Fanuc KAREL source: KT00074.KL

PROGRAM KT00074
%NOLOCKGROUP
VAR
  R1: REAL
  I2: INTEGER
  OUT: REAL
BEGIN
  R1 = 2.0
    I2 = 3
  OUT = R1 * I2
END KT00074
